PROGRAM PRG_AxisControl
VAR
	MC_SetZero_Th1: MC_SetPosition;
	MC_SetZero_Th2: MC_SetPosition;
	MC_Jog_Th1: MC_Jog;
	MC_Jog_Th2: MC_Jog;
	MC_MoveAbsolute_Th1: MC_MoveAbsolute;
	MC_MoveAbsolute_Th2: MC_MoveAbsolute;
END_VAR

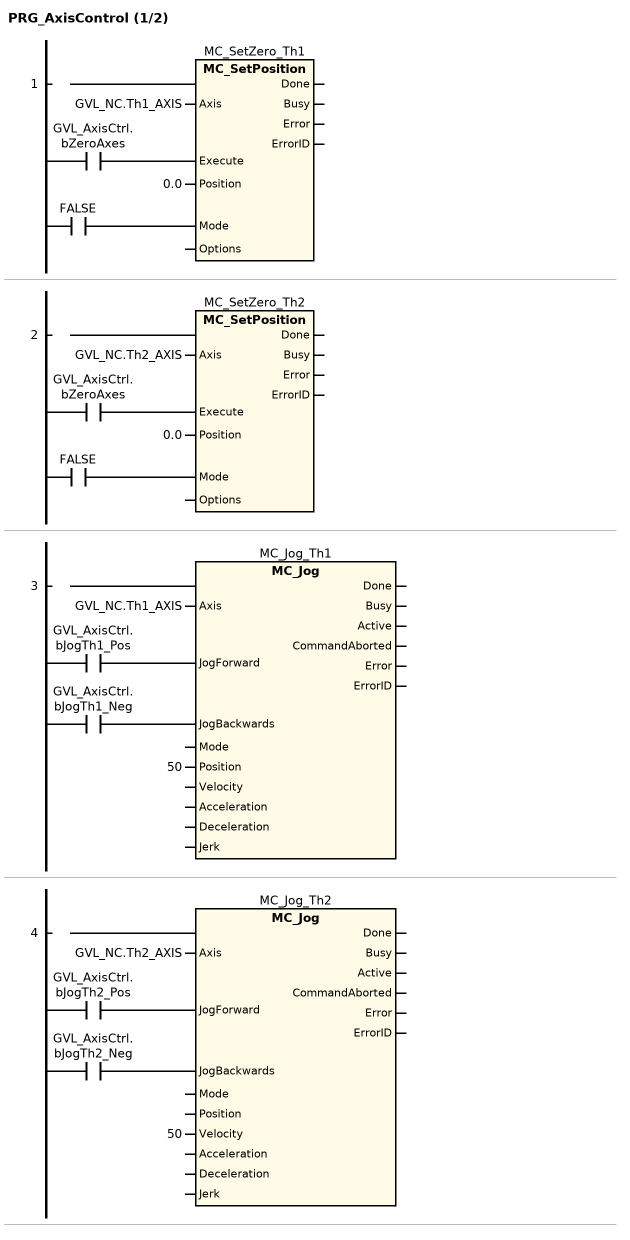
// NETWORK 1
MC_SetZero_Th1(Axis := GVL_NC.Th1_AXIS, Execute := GVL_AxisCtrl.bZeroAxes, Position := 0.0, Mode := FALSE); // MC_SetPosition

// NETWORK 2
MC_SetZero_Th2(Axis := GVL_NC.Th2_AXIS, Execute := GVL_AxisCtrl.bZeroAxes, Position := 0.0, Mode := FALSE); // MC_SetPosition

// NETWORK 3
MC_Jog_Th1(
    Axis := GVL_NC.Th1_AXIS,
    JogForward := GVL_AxisCtrl.bJogTh1_Pos,
    JogBackwards := GVL_AxisCtrl.bJogTh1_Neg,
    Position := 50); // MC_Jog

// NETWORK 4
MC_Jog_Th2(
    Axis := GVL_NC.Th2_AXIS,
    JogForward := GVL_AxisCtrl.bJogTh2_Pos,
    JogBackwards := GVL_AxisCtrl.bJogTh2_Neg,
    Velocity := 50); // MC_Jog

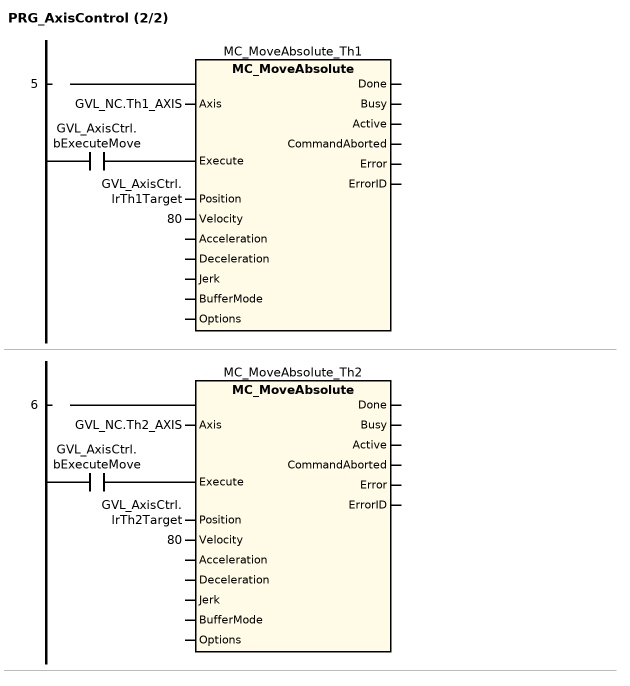
// NETWORK 5
MC_MoveAbsolute_Th1(
    Axis := GVL_NC.Th1_AXIS,
    Execute := GVL_AxisCtrl.bExecuteMove,
    Position := GVL_AxisCtrl.lrTh1Target,
    Velocity := 80); // MC_MoveAbsolute

// NETWORK 6
MC_MoveAbsolute_Th2(
    Axis := GVL_NC.Th2_AXIS,
    Execute := GVL_AxisCtrl.bExecuteMove,
    Position := GVL_AxisCtrl.lrTh2Target,
    Velocity := 80); // MC_MoveAbsolute

END_PROGRAM

(* stored: Version 1.1.0.1, ProductVersion 3.1.4024.2
   POU PRG_AxisControl: Id {80e1f596-e450-427b-95f9-6f95fa895977}, SpecialFunc None *)
